FUNCTION_BLOCK TcSynchronizedAxisCommand IMPLEMENTS itfSynchronizedAxisCommand
VAR_INPUT
END_VAR
VAR_OUTPUT
END_VAR
VAR
END_VAR

{warning 'add method implementation '}
METHOD Abort : MC_Error
END_METHOD

{warning 'add property implementation'}
PROPERTY Active : BOOL
GET
END_GET
END_PROPERTY

{warning 'add property implementation'}
PROPERTY Busy : BOOL
GET
END_GET
END_PROPERTY

{warning 'add property implementation'}
PROPERTY Command : MC_COMMAND_REF
GET
END_GET
END_PROPERTY

{warning 'add property implementation'}
PROPERTY CommandAborted : BOOL
GET
END_GET
END_PROPERTY

{warning 'add property implementation'}
PROPERTY Done : BOOL
GET
END_GET
END_PROPERTY

{warning 'add property implementation'}
PROPERTY Error : BOOL
GET
END_GET
END_PROPERTY

{warning 'add property implementation'}
PROPERTY ErrorId : MC_Error
GET
END_GET
END_PROPERTY

{warning 'add property implementation'}
PROPERTY InSync : BOOL
GET
Insync:= Geared;
END_GET
END_PROPERTY

{warning 'add method implementation '}
METHOD Update 		: MC_Error
VAR_INPUT
	Position		: REAL;
	Velocity		: REAL;
	EndVelocity		: REAL;
	Acceleration	: REAL;
	Deceleration	: REAL;
	Jerk			: REAL;
END_VAR
END_METHOD

{warning 'add method implementation '}
METHOD Wait 		: MC_Error (* This method only makes sense in the IEC 61499 environment*)
VAR_INPUT
	Timeout			: TIME;
	AbortOnTimeout	: BOOL;
END_VAR
END_METHOD

END_FUNCTION_BLOCK

(* stored: Version 1.1.0.1, ProductVersion 3.1.4024.11
   POU TcSynchronizedAxisCommand: Id {5df8cfc3-abf9-40b2-afe9-4ec11a9d63ce}, SpecialFunc None
   Method Abort: Id {1742accd-7e31-4de7-ad6d-abdeb6f6e916}
   Property Active: Id {763c79c4-691f-41e0-a358-3c2dd370d22c}
   Get Get: Id {9ca1fed1-b1bd-4db9-b364-10f5a0c23170}
   Property Busy: Id {99a6c568-eba9-4015-9b86-96a911e34eec}
   Get Get: Id {4e4b59f3-ed21-41f8-8ef7-a8140f8f1499}
   Property Command: Id {47c3cc3a-5f2f-4012-8055-07d3a395ef2b}
   Get Get: Id {cdc4eae6-f25e-4af7-8719-fe7916b77d7d}
   Property CommandAborted: Id {17dbeaab-e4c1-4806-9db3-6655101dc6c6}
   Get Get: Id {df65dcc8-b128-42df-8084-a4391456fae5}
   Property Done: Id {96fc23dd-ff6b-4816-93a9-b6f46a6de6e9}
   Get Get: Id {41e69d85-2cb5-4420-8aac-7e83c7fa7ae1}
   Property Error: Id {d2e0a4a9-2cf6-459e-bac6-8059f81cd70b}
   Get Get: Id {22eb0086-9134-4ae2-a759-eeb8e0905b8d}
   Property ErrorId: Id {782cc100-e1f5-4c50-a541-a7ff82ee610a}
   Get Get: Id {b6321dca-290a-49a5-bc87-bc241efeeabd}
   Property InSync: Id {71bfe119-3f6f-45dc-b508-cb21c2b3c41f}
   Get Get: Id {14856b60-1e6a-481c-ab7e-94b920dd284d}
   Method Update: Id {c3e88328-200d-49ce-81b5-aa2d2fa3f98b}
   Method Wait: Id {72a42516-532d-42c2-9f57-fc368752168f} *)
